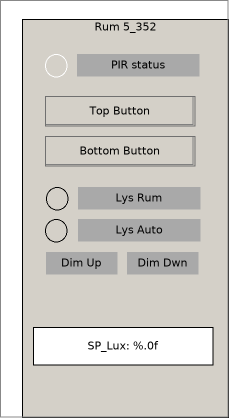
VISUALIZATION Visualization_5_352_1_1_1_1_1_2_1  // 229x418
    RoundedRectangle (22,19 207x399), "Rum 5_352"
    Rectangle (33,327 180x38), "SP_Lux: %.0f", text variable: P_Rum_4_324.fbLys.fbLightCtrl.fLuxZone1
    Button (45,96 150x30), "Top Button"
        tap P_Rum_5_352.bTopButtonZone1_Visu
    Button (45,136 150x30), "Bottom Button"
        tap P_Rum_5_352.bBottomButtonZone1_Visu
    Ellipse (46,187 22x23), colour toggle: P_Rum_5_352.fbLys.fbLightCtrl.bOnZone1
    Rectangle (78,187 122x22), "Lys Rum"
    Rectangle (46,252 71x22), "Dim Up", colour toggle: P_Rum_5_352.fbLys.fbLightCtrl.bDimUp
    Rectangle (127,252 71x22), "Dim Dwn", colour toggle: P_Rum_5_352.fbLys.fbLightCtrl.bDimDwn
    Ellipse (45,219 22x23), colour toggle: P_Rum_5_352.fbLys.fbLightCtrl.bAutoZone1
    Rectangle (78,219 122x22), "Lys Auto"
    Ellipse (45,54 22x23), colour toggle: P_Rum_5_352.fbLys.fbLightCtrl.bPIR
    Rectangle (77,54 122x22), "PIR status"
END_VISUALIZATION

(* stored: Version 1.1.0.1
   Visu Visualization_5_352_1_1_1_1_1_2_1: Id {fe9a7a2b-69eb-4622-a365-42d94a54fc18} *)
